TYPE TcaRackFeederConfig :
STRUCT
END_STRUCT
END_TYPE

(* stored: Version 1.1.0.1
   DUT TcaRackFeederConfig: Id {ef8e05e7-8f38-4e4d-9105-75fb9f1af3ef} *)
